Staubli VAL3: loadmaster1.pgx

program loadmaster1(string x_sMasterFile1 (dimensions=1))
begin
  if master:libLoad(x_sMasterFile1)<0
    popUpMsg("nO ok")
  endIf
  frmaster[1].trsf=master:tTool.trsf
  //取个数
  nsize[1]=size(master:ptRoutingPath)
  //存个数
  resize(pdemo1,1,nsize[1])
  //保存程序
  master:libSave()
end
